(* IEC 61131-3 sources: stc/pkg/analyzer/testdata, 3 files *)

(* ---- multi_file_a.st ---- *)
FUNCTION_BLOCK FB_Motor
VAR_INPUT
    bStart : BOOL;
END_VAR
VAR
    running : BOOL;
END_VAR
    running := bStart;
END_FUNCTION_BLOCK

(* ---- vendor_test.st ---- *)
FUNCTION_BLOCK MyFB
VAR
    counter : INT;
END_VAR

METHOD PUBLIC DoWork : BOOL
VAR_INPUT
    value : INT;
END_VAR
    DoWork := value > 0;
END_METHOD

END_FUNCTION_BLOCK

(* ---- multi_file_b.st ---- *)
PROGRAM Main
VAR
    motor : FB_Motor;
    startFlag : BOOL;
END_VAR
    startFlag := TRUE;
END_PROGRAM
